TYPE
    WrappedComponentExample_Config EXTENDS TcoCore.TcoStruct :
    STRUCT

        VacuumReachedStabilisation : TIME := T#100MS;
        VacuumPushTime : TIME := T#100MS;
    END_STRUCT
END_TYPE

(* stored: Version 1.1.0.1
   DUT WrappedComponentExample_Config: Id {b2440eb9-9624-468f-adb0-1ba14e8f1deb} *)
